// TIA Portal V20 export
DATA_BLOCK "DB_NordSetPoint"   // DB35
// stored: Access Published, MemoryReserve 100, Namespace EmptyLine
   VAR
      Line : Struct
         EmptyLine : Struct   // -(0 - 16000) -> (CW: 0 - 100%) || +(0 - 16000) (CCW: 0 - 100%) || freq. has been set via NORDCON
            Conveyor : Array[_.minEmptyLine.._.maxEmptyLine] of DInt;
         END_STRUCT;
      END_STRUCT;
   END_VAR
BEGIN
END_DATA_BLOCK
